	      //-----------------------------------------------------------------------------
	      // continue motion in SINGLESTEP mode
	      //-----------------------------------------------------------------------------
	      // check for execution to be waiting for new rising edge
	    ELSIF #statStateExecution = #EX_TRIGGERING_CMD
	      AND #statExecutionWaitSingleStep = TRUE
	    THEN
	      #statBusy := TRUE; // set FB state to busy
	      #statExecutionWaitSingleStep := FALSE; // reset execution wait bit stopping cmds from being executed (wait in EX_TRIGGERING_CMD)
	      //===========================================================================================
	      
	      //-----------------------------------------------------------------------------
	      // CONTINUE after interrupt
	      //-----------------------------------------------------------------------------
	      // check for path motion to be interrupted
	    ELSIF #statStateExecution = #EX_INTERRUPTED
	      OR #statStateExecution = #EX_INTERRUPTING // FR 12.10.2021
	    THEN
	      // State machine - continue path motion and sequence
	      // no changes to PreBuffer state machine
	      #statStateExecution := #EX_CONTINUEING;
	      // no setting of FB state to busy necessary, interrupt does not reset busy
	      // ==========================================================================================
	      
	      //-----------------------------------------------------------------------------
	      // RETRIGGER during running path motion
	      //-----------------------------------------------------------------------------
	      // check for path motion to be running with all previous cmds executed
	    ELSIF #statStateExecution = #EX_ALL_TRIGGERED THEN
	      #statBusy := TRUE; // set FB state to busy
	      #statLastCmdIdPathdata := 0; // reset last cmdId in PathData depending on type of attached PathData
	      #statMCExecuteWasDone := FALSE; // Reset bit to memorize done output of MC_ExecuteKinMotionCmd
	      // state machines - reStart processing
	      #statStatePreBuffering := #PB_ENABLED;
	      #statStateExecution := #EX_GET_CMD;
	      // initialize variables
	      #statReadyForNextPath := FALSE;
	      // set status - added JR 2019/04/16
	      #statStatus := #STATUS_SUBSEQUENT_CALL;
	      
	      #instLKinCtrl_PreBuffer.flagLimits.firstFlag := LOWER_BOUND(ARR := #flags, DIM := 1);
	      #instLKinCtrl_PreBuffer.flagLimits.lastFlag := UPPER_BOUND(ARR := #flags, DIM := 1);
	      
	      #instLKinCtrl_PreBuffer.flagLimits.firstValueFlag := LOWER_BOUND(ARR := #valueFlags, DIM := 1);
	      #instLKinCtrl_PreBuffer.flagLimits.lastValueFlag := UPPER_BOUND(ARR := #valueFlags, DIM := 1);
	      
	      #instLKinCtrl_MC_ExecuteKinMotionCmd.flagLimits.firstFlag := LOWER_BOUND(ARR := #flags, DIM := 1);
	      #instLKinCtrl_MC_ExecuteKinMotionCmd.flagLimits.lastFlag := UPPER_BOUND(ARR := #flags, DIM := 1);
	      
	      #instLKinCtrl_MC_ExecuteKinMotionCmd.flagLimits.firstValueFlag := LOWER_BOUND(ARR := #valueFlags, DIM := 1);
	      #instLKinCtrl_MC_ExecuteKinMotionCmd.flagLimits.lastValueFlag := UPPER_BOUND(ARR := #valueFlags, DIM := 1);
	      
	      //===========================================================================================
	      
	      //-----------------------------------------------------------------------------
	      // START of path motion (initial)
	      //-----------------------------------------------------------------------------
	      // check for path motion not to be running already
	    ELSIF #tempMotionQueueCommands = 0                      // no commands in MotionQueue
	      AND #tempKinematicsStatusWord.%X12 = TRUE             // TO Kinematics in constant velocity
	      AND #axesGroup.StatusPath.Velocity = 0.0              // TO Kinematics standing still
	      AND (#tempKinematicsStatusWord.%X6                    // no motion job in progress
	      OR #axesGroup.StatusConveyor[1].TrackingState <> 0    // If kinematics is in tracking then done (.X6) is not set
	      OR #axesGroup.StatusConveyor[2].TrackingState <> 0
	      OR #axesGroup.StatusConveyor[3].TrackingState <> 0)
	      AND #statStatus <> #STATUS_EXECUTION_WAITING          // Added FR 2019.03.28
	    THEN
	      // Initialize variables, diagnostics, etc.
	      #statStatus := #STATUS_FIRST_CALL;
	      #statStateExecution := #EX_RESETTING;
	      
	      #instLKinCtrl_PreBuffer.flagLimits.firstFlag := LOWER_BOUND(ARR := #flags, DIM := 1);
	      #instLKinCtrl_PreBuffer.flagLimits.lastFlag := UPPER_BOUND(ARR := #flags, DIM := 1);
	      
	      #instLKinCtrl_PreBuffer.flagLimits.firstValueFlag := LOWER_BOUND(ARR := #valueFlags, DIM := 1);
	      #instLKinCtrl_PreBuffer.flagLimits.lastValueFlag := UPPER_BOUND(ARR := #valueFlags, DIM := 1);
	      
	      #instLKinCtrl_MC_ExecuteKinMotionCmd.flagLimits.firstFlag := LOWER_BOUND(ARR := #flags, DIM := 1);
	      #instLKinCtrl_MC_ExecuteKinMotionCmd.flagLimits.lastFlag := UPPER_BOUND(ARR := #flags, DIM := 1);
	      
	      #instLKinCtrl_MC_ExecuteKinMotionCmd.flagLimits.firstValueFlag := LOWER_BOUND(ARR := #valueFlags, DIM := 1);
	      #instLKinCtrl_MC_ExecuteKinMotionCmd.flagLimits.lastValueFlag := UPPER_BOUND(ARR := #valueFlags, DIM := 1);
	      //===========================================================================================
	      
	    ELSE
	      //===========================================================================================
	      // Trigger not possible
	      // set execution state machine
	      #statStateExecution := #EX_ERROR_STATE;
	      #statStatus := #ERR_TRIGGER_NOT_POSSIBLE;
	      //===========================================================================================
	    END_IF;
	    
	  ELSIF (#statStatus = #STATUS_FIRST_CALL) THEN
	    #statStatus := #STATUS_SUBSEQUENT_CALL;
	  END_IF;
	  
	  // Edge detection input variables
	  #statExecuteOld := #tempExecute;
	  #statStopOld := #tempStop;
	  #statInterruptOld := #tempInterrupt;
	  #statResetOld := #tempReset;
	  
	END_REGION TRIGGERING
	
	IF (#statStatus = #STATUS_NO_CALL) THEN // Nothing to do -> End here to reduce "system load"
	  RETURN;
	END_IF;
	
	REGION RESETTING
	  IF #statStateExecution = #EX_RESETTING
	    // AND #statDebugState = TRUE
	  THEN
	    // reset  variable for single step debugging of states
	    #statDebugState := FALSE;
	    
	    // ----------------------------------------------
	    // Reset static for outputs
	    // ----------------------------------------------
	    #statDone := FALSE;
	    #statCommandAborted := FALSE;
	    #statError := FALSE;
	    #statErrorID := 16#0;
	    #statSubfunctionStatus := 16#0;
	    #diagnostics := #statEmptyDiagnostics;
	    
	    // ----------------------------------------------
	    // reset static variables
	    //-----------------------------------------------
	    #statFirstCycle := TRUE;
	    #statInterruptedAtStart := FALSE;
	    #statExecutionWaitSingleStep := FALSE;
	    #statPauseExecution := FALSE;
	    #statMCExecuteWasDone := FALSE;
	    #statPathDataIdentifier := 0;
	    #statLastCmdIdPathdata := 0;
	    #statWrittenActiveCmdNo := -1;
	    #statStoreInterruptStateExecution := 0;
	    #statPreBufferCmdCtr := "LKINCTRL_NO_OF_START_EXECUTE_CMDS";
	    #statAbortOld := FALSE;
	    #statIsMeasurementCmd := 0;
	    
	    
	    // ----------------------------------------------
	    // initialize buffer variables
	    //-----------------------------------------------
	    // Reset PathDataPreBuffered
	    #statPathDataElementPreBuffered := #statEmptyPathDataElementPreBuffered;
	    FOR #tempCtr := 1 TO "LKINCTRL_NO_OF_PATHDATA_PREBUFFER_ELEMENTS" DO
	      #statPathDataPreBuffered.commands[#tempCtr] := #statEmptyPathDataElementPreBuffered;
	    END_FOR;
	    #statPathDataPreBuffered.retrievePointer := 1;
	    #statPathDataPreBuffered.addPointer := 1;
	    #statPathDataPreBuffered.addPointerRestarted := FALSE;
	    #statPathDataPreBuffered.pathDataName := '';
	    #statPathDataPreBufferAddPointerOld := 0;
	    
	    // ----------------------------------------------
	    // initialize flag handling variables
	    //-----------------------------------------------
	    // Reset waitFlags struct
	    #statWaitFlags.waitCtr := 0;
	    FOR #tempCtr := 1 TO "LKINCTRL_NO_OF_CMD_SETFLAGS" DO
	      #statWaitFlags.waitFlag[#tempCtr] := -1;
	    END_FOR;
	    
	    // Reset waitValueFlag struct
	    #statWaitValueFlags.waitCtr := 0;
	    FOR #tempCtr := 1 TO "LKINCTRL_NO_OF_CMD_VALUEFLAGS" DO
	      #statWaitValueFlags.waitFlag[#tempCtr] := -1;
	    END_FOR;
	    
	    // Reset setFlagsBuffer variables
	    #statFlagsBuffer.writeBufferElement := 1;
	    #statSetFlagsBufferWriteBufferElement_old := 1;
	    
	    // Reset setFlagBuffer
	    FOR #tempCtr := 1 TO "LKINCTRL_NO_OF_SETFLAGS_BUFFER_ELEMENTS" DO
	      #statFlagsBuffer.bufferElement[#tempCtr] := #statEmptyFlagBufferElement;
	    END_FOR;
	    
	    // ----------------------------------------------
	    // Call instances with false
	    // ----------------------------------------------
	    #instLKinCtrl_MC_ExecuteKinMotionCmd(execute                 := FALSE,
	                                         interrupt               := FALSE,
	                                         continueMotion          := FALSE,
	                                         stopMode                := #configuration.stopMode,
	                                         interruptMode           := #configuration.interruptMode,
	                                         reset                   := FALSE,
	                                         stop                    := FALSE,
	                                         writtenActiveCmdNo      := #statWrittenActiveCmdNo,
	                                         conveyorConfiguration   := #configuration.conveyorParameter,
	                                         userFrames              := #configuration.userFrames,
	                                         workspaceZones          := #configuration.workspaceZones,
	                                         kinematicsZones         := #configuration.kinematicsZones,
	                                         pauseCmdExecution       => #statPauseExecution,
	                                         activePathDataName      => #statActivePathData,
	                                         activeCmdNo             => #statActiveCmdNo,
	                                         remainingDistanceActCmd => #statRemainingDistanceActCmd,
	                                         activeUserFrames        => #activeUserFrames,
	                                         pathDataElementPreBuf   := #statPathDataElementPreBuffered,
	                                         to_Kinematics           := #axesGroup);
	    
	    IF #statStatus = #STATUS_FB_RESETTING
	      OR #statStatus = #STATUS_FIRST_CALL
	    THEN
	      #instLKinCtrl_MC_ExecuteKinMotionCmd.reset := TRUE; // If resetting then also reset MC_ExecuteKinMotionCmd
	      #instLKinCtrl_MC_ExecuteKinMotionCmd(execute                 := FALSE,
	                                           interrupt               := FALSE,
	                                           continueMotion          := FALSE,
	                                           stopMode                := #configuration.stopMode,
	                                           interruptMode           := #configuration.interruptMode,
	                                           //reset := FALSE, // written above
	                                           stop                    := FALSE,
	                                           writtenActiveCmdNo      := #statWrittenActiveCmdNo,
	                                           conveyorConfiguration   := #configuration.conveyorParameter,
	                                           userFrames              := #configuration.userFrames,
	                                           workspaceZones          := #configuration.workspaceZones,
	                                           kinematicsZones         := #configuration.kinematicsZones,
	                                           pauseCmdExecution       => #statPauseExecution,
	                                           activePathDataName      => #statActivePathData,
	                                           activeCmdNo             => #statActiveCmdNo,
	                                           remainingDistanceActCmd => #statRemainingDistanceActCmd,
	                                           activeUserFrames        => #activeUserFrames,
	                                           pathDataElementPreBuf   := #statPathDataElementPreBuffered,
	                                           to_Kinematics           := #axesGroup);
	      #instLKinCtrl_MC_ExecuteKinMotionCmd.reset := FALSE; // Reset input
	    END_IF;
	    
	    #instLKinCtrl_PreBuffer(enable         := FALSE,
	                            error          => #statPreBufferError,
	                            pointTable     := #pointTable,
	                            to_Kinematics  := #axesGroup,
	                            pathData       := #pathData,
	                            pathDataPreBuf := #statPathDataPreBuffered);
	    
	    #instLKinCtrl_SetFlagCtrl(enable    := FALSE,
	                              waitMain  => #statWaitMain,
	                              flags     := #flags,
	                              waitFlags := #statWaitFlags);
	    
	    #instLKinCtrl_ValueFlagCtrl(enable     := FALSE,
	                                waitMain   => #statWaitValueMain,
	                                valueFlags := #valueFlags,
	                                waitFlags  := #statWaitValueFlags);
	    
	    // ----------------------------------------------
	    // Check if coming from reset or execute and handle differences
	    // ----------------------------------------------
	    IF #statStatus = #STATUS_FB_RESETTING THEN
	      // ---------------------------
	      // Coming from reset
	      // ---------------------------
	      #statReadyForNextPath := TRUE;
	      #statStateExecution := #EX_NO_PROCESSING;
	      #statStatePreBuffering := #PB_NO_PROCESSING;
	      #statStatus := #STATUS_NO_CALL;
	    ELSE
	      // ---------------------------
	      // Coming from execute
	      // ---------------------------
	      #statBusy := TRUE;
	      #statReadyForNextPath := FALSE;
	      #statStatePreBuffering := #PB_ENABLED;
	      IF #INTERRUPT_AT_START THEN
	        #statStateExecution := #EX_INTERRUPT_AT_START;
	      ELSIF #CONTINUE_AT_START THEN
	        #statStateExecution := #EX_CONTINUE_AT_START;
	      ELSE
	        #statStateExecution := #EX_GET_CMD;
	      END_IF;
	    END_IF;
	  END_IF;
	END_REGION RESETTING
	
	REGION ABORT_MEASUREMENT_CMD
	  //------------------------------------------------------------------------------------------
	  // Abort measurement command functionality 
	  //------------------------------------------------------------------------------------------
	  //check cyclically if abort input has been reset
	  IF (#statAbortOld = TRUE) AND (#tempAbortMeasurementCmd = FALSE) THEN
	    #statAbortOld := FALSE;
	    
	    //first call of abort functionality
	  ELSIF (#tempAbortMeasurementCmd = TRUE) AND (#statAbortOld = FALSE) THEN
	    IF ((#statIsMeasurementCmd = "LKINCTRL_MEAS_CMD_WO_ACK")
	      OR (#statIsMeasurementCmd = "LKINCTRL_MEAS_CMD_WITH_ACK"))
	    THEN
	      #statActiveCmdNoOld := #statActiveCmdNo;
	      #statStateOld := #statStateExecution;
	      #statStateExecution := #EX_ABORT_MEAS_CMD;
	      #statAbortOld := TRUE;
	    END_IF;
	    
	    //for multiple measurement commands in a row (1,1,1 or 1,1,1,2)
	  ELSIF (#tempAbortMeasurementCmd = TRUE) AND (#statAbortOld = TRUE) THEN
	    IF ((#statIsMeasurementCmd = "LKINCTRL_MEAS_CMD_WO_ACK") OR (#statIsMeasurementCmd = "LKINCTRL_MEAS_CMD_WITH_ACK"))
	      AND (#statActiveCmdNo = (#statActiveCmdNoOld + 1))
	    THEN
	      #statActiveCmdNoOld := #statActiveCmdNo;
	      #statStateOld := #statStateExecution;
	      #statStateExecution := #EX_ABORT_MEAS_CMD;
	      #statAbortOld := TRUE;
	    END_IF;
	  END_IF;
	END_REGION
	
	REGION PRE_BUFFERING
	  
	  // state reached when no pre buffering is active
	  REGION PB_NO_PROCESSING
	    IF #statStatePreBuffering = #PB_NO_PROCESSING
	      // AND #statDebugState = TRUE
	    THEN
	      // reset  variable for single step debugging of states
	      #statDebugState := FALSE;
	      
	      // Do nothing here
	    END_IF;
	  END_REGION PB_NO_PROCESSING
	  
	  // state reached when pre buffering is active
	  REGION PB_ENABLED
	    IF #statStatePreBuffering = #PB_ENABLED
	      // AND #statDebugState = TRUE
	    THEN
	      // reset  variable for single step debugging of states
	      #statDebugState := FALSE;
	      
	      IF #statStatus = #STATUS_FIRST_CALL THEN
	        #statInitStartPos := TRUE;
	      END_IF;
	      
	      
	      // Call FB PreBuffer multiple times
	      FOR #tempCtr := 1 TO #statPreBufferCmdCtr DO
	        
	        // Call FB PreBuffer
	        #instLKinCtrl_PreBuffer(enable                  := TRUE,
	                                initPathTransition      := #pathTransition,
	                                initBufferMode          := #bufferMode,
	                                initTransitionParameter := #transitionParameter,
	                                initStartPosition       := #statInitStartPos,
	                                configuration           := #configuration,
	                                error                   => #statPreBufferError,
	                                pointTable              := #pointTable,
	                                to_Kinematics           := #axesGroup,
	                                lastCmdIdPathData       => #statLastCmdIdPathdata,
	                                pathData                := #pathData,
	                                pathDataPreBuf          := #statPathDataPreBuffered);
	        
	        #statInitStartPos := FALSE;
	        
	        // check for FB PreBuffer to signalize an error
	        IF #statPreBufferError THEN
	          IF #instLKinCtrl_MC_ExecuteKinMotionCmd.busy THEN
	            #statStatus := #STATUS_STOP_DUE_TO_ERROR; // Error at command --> Stop Kinematics
	          ELSE
	            #statStatus := #ERR_PATHDATA_PARAMETERS;
	          END_IF;
	          #statSubfunctionStatus := #instLKinCtrl_PreBuffer.status;// Store subfunction status
	          #statStatePreBuffering := #PB_DISABLED; // Disable preBuffer
	          #statStateExecution := #EX_ERROR_STATE;
	          // Write diagnostics
	          #diagnostics.pathDataName := #statPathDataPreBuffered.pathDataName;
	          #diagnostics.cmdNumber := #instLKinCtrl_PreBuffer.pathDataRetrievePointer;
	          EXIT; // exit loop to end pre buffering
	        END_IF;
	        
	        // Check for FB PreBuffer to have buffered the last element of the PathData to PathData_PreBuf
	        IF #instLKinCtrl_PreBuffer.status = 16#7100 THEN // STATUS_ALL_CMDS_BUFFERED
	          #statStatePreBuffering := #PB_DISABLED; // go to disable state when PreBuffer is done
	          EXIT; // exit loop to end pre buffering
	        END_IF;
	        
	      END_FOR;
	    END_IF;
	  END_REGION PB_ENABLED
	  
	  // state reached when pre buffering is active
	  REGION PB_DISABLED
	    IF #statStatePreBuffering = #PB_DISABLED
	      // AND #statDebugState = TRUE
	    THEN
	      // reset  variable for single step debugging of states
	      #statDebugState := FALSE;
	      
	      // call FB_PreBuffer with false
	      // second call of FB necessary, for PathData with one command only ==> handled in one cycle only
	      #instLKinCtrl_PreBuffer(enable         := FALSE,
	                              pointTable     := #pointTable,
	                              to_Kinematics  := #axesGroup,
	                              pathData       := #pathData,
	                              pathDataPreBuf := #statPathDataPreBuffered);
	      
	    END_IF;
	  END_REGION PB_DISABLED
	  
	END_REGION PRE_BUFFERING
	
	
	REGION EXECUTION
	  // Call Execution steps multiple times
	  FOR #tempExecCtr := 1 TO #statPreBufferCmdCtr DO
	    
	    
	    // state reached when no processing is active 
	    REGION EX_NO_PROCESSING
	      IF #statStateExecution = #EX_NO_PROCESSING
	        // AND #statDebugState = TRUE
	      THEN
	        // reset  variable for single step debugging of states
	        #statDebugState := FALSE;
	        
	        // do nothing and wait for execute trigger
	      END_IF;
	    END_REGION EX_NO_PROCESSING
	    
	    REGION EX_INTERRUPT_AT_START
	      IF #statStateExecution = #EX_INTERRUPT_AT_START THEN
	        #instLKinCtrl_MC_ExecuteKinMotionCmd.interrupt := TRUE; // Simulate interrupt input
	        
	        IF #instLKinCtrl_MC_ExecuteKinMotionCmd.diagnostics.status = 16#7102 THEN // Check if interrupted
	          // Interrupted --> Start executing commands
	          #instLKinCtrl_MC_ExecuteKinMotionCmd.interrupt := FALSE;
	          #statInterruptedAtStart := TRUE;
	          #statStateExecution := #EX_GET_CMD;
	        END_IF;
	      END_IF;
	    END_REGION EX_INTERRUPT_AT_START
	    
	    REGION EX_CONTINUE_AT_START
	      // Due to a system bug up to FW4.0 (blending, override) a groupContinue must always be triggered after a groupInterrupt even if the interrupt was aborted with a groupStop.
	      // To avoid checking for aborted interrupts we always trigger continue at the start of a path.
	      IF #statStateExecution = #EX_CONTINUE_AT_START THEN
	        IF #tempKinematicsStatusWord.%X17 = FALSE THEN // Only continue if not interrupted as we dont want to trigger a movement
	          #instLKinCtrl_MC_ExecuteKinMotionCmd.continueMotion := TRUE; // Trigger continue
	          
	          IF #instLKinCtrl_MC_ExecuteKinMotionCmd.diagnostics.status = 16#7100 THEN // Check if continue is done
	            #instLKinCtrl_MC_ExecuteKinMotionCmd.continueMotion := FALSE;
	            #statStateExecution := #EX_GET_CMD;
	          END_IF;
	        ELSE
	          // Go to next step if interrupted from extern
	          #statStateExecution := #EX_GET_CMD;
	        END_IF;
	      END_IF;
	    END_REGION EX_CONTINUE_AT_START
	    
	    // state reached new command should be provided from PathData_PreBuffered to LKinCtrl_ExecuteKinMotionCmd 
	    REGION EX_GET_CMD
	      IF #statStateExecution = #EX_GET_CMD
	        // AND #statDebugState = TRUE
	      THEN
	        // reset  variable for single step debugging of states
	        #statDebugState := FALSE;
	        #statSubfunctionStatus := 16#0;
	        
	        // check for lastCmdIdPathInData to be recognized after last execution of EX_TRIGGERED_CMD
	        IF #statPathDataElementPreBuffered.cmdID = #statLastCmdIdPathdata
	          AND #statPathDataElementPreBuffered.isIntermediateCmd = FALSE
	        THEN
	          // skip GET_NEW_CMD and go to EX_ALL_TRIGGERED
	          #statStateExecution := #EX_ALL_TRIGGERED;
	        ELSE
	          // ------------------------------------------------------------------------------------------
	          // Get new cmd from PathData_PreBuffered according to the pointer status
	          // ------------------------------------------------------------------------------------------
	          // Initialize temp
	          #tempPreBufferPtrOk := FALSE;
	          
	          // Check if addPointer was restarted 
	          IF #statPathDataPreBuffered.addPointerRestarted THEN
	            // addPointer must not pass retrievePointer (no overwriting not read slots), addPointer may not pass
	            #tempPreBufferPtrOk := #statPathDataPreBuffered.retrievePointer > #statPathDataPreBuffered.addPointer;
	            
	            // Special cases in first cycle or contourOffset and addPointerRestarted
	            IF #statStatus = #STATUS_FIRST_CALL OR #instLKinCtrl_PreBuffer.preBufferLockDueToConfigCmd THEN
	              #tempPreBufferPtrOk := TRUE;
	            END_IF;
	          ELSE
	            // retrievePointer must not pass addPointer (no reading of empty slots), retrievePointer may not pass
	            #tempPreBufferPtrOk := #statPathDataPreBuffered.retrievePointer < #statPathDataPreBuffered.addPointer;
	          END_IF;
	          
	          IF #tempPreBufferPtrOk THEN
	            // ------------------------------------------------------------------------------------------
	            // Copy command for execution and increase retrievePointer
	            // ------------------------------------------------------------------------------------------
	            #statPathDataElementPreBuffered := #statPathDataPreBuffered.commands[#statPathDataPreBuffered.retrievePointer];
	            
	            // Calculate new retrievePointer
	            IF #statPathDataPreBuffered.retrievePointer < "LKINCTRL_NO_OF_PATHDATA_PREBUFFER_ELEMENTS" THEN
	              #statPathDataPreBuffered.retrievePointer += 1;
	            ELSE
	              #statPathDataPreBuffered.retrievePointer := 1;  // restart PathDataPreBuf retrievePointer
	              #statPathDataPreBuffered.addPointerRestarted := FALSE; // reset restart bit of pointer
	            END_IF;
	            
	            // ------------------------------------------------------------------------------------------
	            // PathData identifier number - setting
	            // ------------------------------------------------------------------------------------------
	            // detect change of PathData - new cmdId smaller or equal to last one ==> new Path
	            IF (#statPathDataElementPreBuffered.cmdID <= #statPreBufferedCmdIdOld)
	              OR (#statPathDataElementPreBuffered.pathDataName <> #statPreBufferedPathDataNameOld)
	            THEN
	              // handle PathData identifier counter
	              IF #statPathDataIdentifier < "LKINCTRL_NO_OF_SETFLAGS_BUFFER_ELEMENTS" THEN
	                #statPathDataIdentifier += 1; // increase PathData counter
	              ELSE
	                #statPathDataIdentifier := 1; // restart PathData identifier counter
	              END_IF;
	            END_IF;
	            
	            // write PathData identifier in PatDataElement_preBuffered
	            #statPathDataElementPreBuffered.pathDataIdentifier := #statPathDataIdentifier;
	            
	            // store old cmdID and PathDataName
	            #statPreBufferedCmdIdOld := #statPathDataElementPreBuffered.cmdID;
	            #statPreBufferedPathDataNameOld := #statPathDataElementPreBuffered.pathDataName;
	            
	            
	            // ------------------------------------------------------------------------------------------
	            // FLAG information - store and evaluate
	            // ------------------------------------------------------------------------------------------
	            // copy command setFlags for storing and usage in flag handling
	            // setFlagsBuffer has twice the number of slots of PathDataPreBuffered to store flag information of past executed (already in MotionQueue) commands
	            #tempFlagBufferElement.pathDataName := #statPathDataElementPreBuffered.pathDataName;
	            #tempFlagBufferElement.pathDataIdentifier := #statPathDataIdentifier;
	            #tempFlagBufferElement.cmdId := #statPathDataElementPreBuffered.cmdID;
	            #tempFlagBufferElement.setFlags := #statPathDataElementPreBuffered.setFlags;
	            #tempFlagBufferElement.valueFlags := #statPathDataElementPreBuffered.valueFlags;
	            #tempFlagBufferElement.isIntermediateCmd := #statPathDataElementPreBuffered.isIntermediateCmd;
	            
	            #statFlagsBuffer.bufferElement[#statFlagsBuffer.writeBufferElement] := #tempFlagBufferElement;
	            
	            #statSetFlagsBufferWriteBufferElement_old := #statFlagsBuffer.writeBufferElement;
	            
	            // increase statSetFlagsBuffer write pointer and restart at overflow
	            IF #statFlagsBuffer.writeBufferElement < "LKINCTRL_NO_OF_SETFLAGS_BUFFER_ELEMENTS" THEN
	              #statFlagsBuffer.writeBufferElement := #statFlagsBuffer.writeBufferElement + 1;
	            ELSE
	              #statFlagsBuffer.writeBufferElement := 1;
	            END_IF;
	            
	            // ------------------------------------------------------------------------------------------
	            // Go to next state --> Trigger command
	            // ------------------------------------------------------------------------------------------
	            #statStateExecution := #EX_TRIGGERING_CMD;
	            
	          ELSE
	            // ------------------------------------------------------------------------------------------
	            // PreBuffer Pointer do not allow for next command
	            // ------------------------------------------------------------------------------------------ 
	            // set subfunction status according to PreBuffer status
	            IF (#statPathDataPreBuffered.retrievePointer = #statPathDataPreBuffered.addPointer
	              AND #statPathDataPreBuffered.addPointerRestarted = FALSE)
	            THEN
	              #statSubfunctionStatus := #STATUS_WAITING_FOR_PREBUFFERED_CMD;
	              
	            ELSIF (#statPathDataPreBuffered.addPointerRestarted = TRUE
	              AND (#statPathDataPreBuffered.retrievePointer - 1 = #statPathDataPreBuffered.addPointer))
	            THEN
	              #statSubfunctionStatus := #STATUS_PREBUFFERED_FULL;
	            END_IF;
	            
	          END_IF;
	          
	          // ------------------------------------------------------------------------------------------
	          // Check if interrupt was executed at start and if continue is needed
	          // ------------------------------------------------------------------------------------------
	          IF #statInterruptedAtStart THEN
	            IF #tempMotionQueueCommands >= MIN(IN1 := #NO_OF_COMMANDS_PRELOADING, IN2 := #axesGroup.MotionQueue.MaxNumberOfCommands)
	              OR #statPauseExecution // Continue if FB ExecuteKinMotionCmd signalizes pause else we have a deadlock
	              OR #statPathDataElementPreBuffered.cmdID = #statLastCmdIdPathdata // Continue if end of path was reached
	            THEN
	              #statStoreInterruptStateExecution := #statStateExecution;
	              #statStateExecution := #EX_CONTINUEING;
	              #statInterruptedAtStart := FALSE;
	            END_IF;
	          END_IF;
	        END_IF;
	      END_IF;
	    END_REGION EX_GET_CMD
	    
	    
	    // state reached when cmd should be triggered
	    REGION EX_TRIGGERING_CMD
	      IF #statStateExecution = #EX_TRIGGERING_CMD
	        // AND #statDebugState = TRUE
	      THEN
	        // Reset variable for single step debugging of states
	        #statDebugState := FALSE;
	        
	        // Create condition for execution
	        #tempExecutionWaiting := #statExecutionWaitSingleStep OR #statPauseExecution OR #statWaitMain OR #statWaitValueMain;
	        
	        IF #tempExecutionWaiting = FALSE THEN
	          // ------------------------------------------------------------------------------------------
	          // Trigger FB_ExecutePathMotion to execute cmd in same cycle
	          // ------------------------------------------------------------------------------------------ 
	          #instLKinCtrl_MC_ExecuteKinMotionCmd.execute := TRUE;
	        ELSIF #instLKinCtrl_MC_ExecuteKinMotionCmd.active = FALSE AND #statStatus <> #STATUS_CMD_CONFIGURATION_ACTIVE AND #tempMotionQueueCommands = 0 THEN
	          // ------------------------------------------------------------------------------------------ 
	          // Execution is waiting
	          // ------------------------------------------------------------------------------------------  
	          #statStatus := #STATUS_EXECUTION_WAITING;
	        ELSE
	          ;
	        END_IF;
	      END_IF;
	    END_REGION EX_TRIGGERING_CMD
	    
	    // state reached when GroupInterrupt is interrupted ==> do nothing when interrupted
	    REGION EX_CONTINUEING
	      IF #statStateExecution = #EX_CONTINUEING
	        // AND #statDebugState = TRUE
	      THEN
	        // reset  variable for single step debugging of states
	        #statDebugState := FALSE;
	        
	        // FR 14.12.2021: Switched IF and trigger to at least have one cycle where continueMotion is true
	        
	        // set state machine to CONTINUED after successfull continue of path motion
	        IF #instLKinCtrl_MC_ExecuteKinMotionCmd.diagnostics.status = 16#7100 // Motion was continued
	          OR (#statMCExecuteWasDone = TRUE AND #instLKinCtrl_MC_ExecuteKinMotionCmd.continueMotion = TRUE) // Motion was done but continue was triggered at least for one cycle
	        THEN
	          #statStateExecution := #EX_CONTINUED;
	        END_IF;
	        
	        // set continueMotion input on LKinCtrl_ExecuteKinMotionCmd
	        // FR 12.10.2021
	        #instLKinCtrl_MC_ExecuteKinMotionCmd.execute := FALSE; // Reset execute
	        #instLKinCtrl_MC_ExecuteKinMotionCmd.continueMotion := TRUE; // Trigger continue
	        #instLKinCtrl_MC_ExecuteKinMotionCmd.interrupt := FALSE; // Reset interrupt
	        
	      END_IF;
	    END_REGION EX_CONTINUEING
	    
	    
	    // state reached when GroupContinue is done ==> do nothing when path motion continues
	    REGION EX_CONTINUED
	      IF #statStateExecution = #EX_CONTINUED
	        // AND #statDebugState = TRUE
	      THEN
	        // reset  variable for single step debugging of states
	        #statDebugState := FALSE;
	        
	        #instLKinCtrl_MC_ExecuteKinMotionCmd.continueMotion := FALSE; // reset continueMotion input on LKinCtrl_ExecuteKinMotionCmd
	        #statStatus := #STATUS_PATHMOTION_RUNNING; // set status accordingly
	        #statStateExecution := #statStoreInterruptStateExecution; // set state machine to state before interrupt
	      END_IF;
	    END_REGION EX_CONTINUED
	    
	    // state reached to execute MC_GroupInterrupt ==> wait for interrupt to be done
	    REGION EX_INTERRUPTING
	      IF #statStateExecution = #EX_INTERRUPTING
	        // AND #statDebugState = TRUE
	      THEN
	        // reset  variable for single step debugging of states
	        #statDebugState := FALSE;
	        
	        #instLKinCtrl_MC_ExecuteKinMotionCmd.execute := FALSE; // Reset execute
	        #instLKinCtrl_MC_ExecuteKinMotionCmd.continueMotion := FALSE; // FR 11.03.2020: Also reset continue input
	        #instLKinCtrl_MC_ExecuteKinMotionCmd.interrupt := TRUE; // Trigger interrupt
	        
	        // check for path motion to have been interrupted (by LKinCtrlExecuteKinMotionCmd)
	        IF #instLKinCtrl_MC_ExecuteKinMotionCmd.diagnostics.status = 16#7102 THEN
	          #statStateExecution := #EX_INTERRUPTED;
	        END_IF;
	      END_IF;
	    END_REGION EX_INTERRUPTING
	    
	    
	    // state reached when path motion has been interrupted in LKinExectuteKinMotionCmd
	    REGION EX_INTERRUPTED
	      IF #statStateExecution = #EX_INTERRUPTED
	        // AND #statDebugState = TRUE
	      THEN
	        // reset variable for single step debugging of states
	        #statDebugState := FALSE;
	        
	        #instLKinCtrl_MC_ExecuteKinMotionCmd.interrupt := FALSE; // Reset interrupt input
	        #statStatus := #STATUS_PATHMOTION_INTERRUPTED; // set status accordingly
	      END_IF;
	    END_REGION EX_INTERRUPTED
	    
	    REGION EX_ABORT_MEAS_CMD
	      IF #statStateExecution = #EX_ABORT_MEAS_CMD
	        //AND #statDebugState = TRUE
	      THEN
	        //abort command
	        #tempStopMeasure := TRUE;
	        #instLKinCtrl_MC_ExecuteKinMotionCmd.execute := FALSE; // Reset execute
	        #instLKinCtrl_MC_ExecuteKinMotionCmd.continueMotion := FALSE; // Reset continue input
	        #instLKinCtrl_MC_ExecuteKinMotionCmd.interrupt := FALSE; // Reset interrupt
	        
	        #statStatus := #STATUS_PATHMOTION_STOPPING; // set status accordingly
	        
	        IF #instLKinCtrl_MC_ExecuteKinMotionCmd.commandAborted THEN // check for path motion to be aborted in LKinExectuteKinMotionCmd
	          #statStateExecution := #EX_MEAS_CMD_ABORTED;
	          #tempStopMeasure := FALSE;
	        ELSIF #instLKinCtrl_MC_ExecuteKinMotionCmd.diagnostics.status.%X15 THEN // check for executer status >= 16#8000
	          #statStateExecution := #EX_ERROR_STATE;
	          #statStatus := #ERR_EXECUTE_KINMOTIONCMD;
	          #statSubfunctionStatus := #instLKinCtrl_MC_ExecuteKinMotionCmd.diagnostics.status;
	        END_IF;
	        
	      END_IF;
	    END_REGION EX_ABORT_MEAS_CMD
	    
	    REGION EX_MEAS_CMD_ABORTED
	      IF #statStateExecution = #EX_MEAS_CMD_ABORTED THEN
	        //if abort signal has to be acknowledged in order to continue
	        IF #statIsMeasurementCmd = "LKINCTRL_MEAS_CMD_WITH_ACK" THEN
	          IF #tempAbortMeasurementCmd = FALSE THEN
	            #statAbortOld := FALSE;
	            #statStateExecution := #statStateOld;
	            IF #statStateExecution = #EX_ALL_TRIGGERED THEN
	              #statMCExecuteWasDone := TRUE;
	            END_IF;
	          END_IF;
	        ELSIF #statIsMeasurementCmd = "LKINCTRL_MEAS_CMD_WO_ACK" THEN
	          #statStateExecution := #statStateOld;
	          IF #statStateExecution = #EX_ALL_TRIGGERED THEN
	            #statMCExecuteWasDone := TRUE;
	          END_IF;
	          IF #tempAbortMeasurementCmd = FALSE THEN
	            #statAbortOld := FALSE;
	          END_IF;
	        END_IF;
	      END_IF;
	    END_REGION EX_MEAS_CMD_ABORTED
	    
	    // state reached when stop input is triggered (path motion stop is executed in LKinExectuteKinMotionCmd)
	    REGION EX_STOPPING
	      IF #statStateExecution = #EX_STOPPING
	        // AND #statDebugState = TRUE
	      THEN
	        // reset variable for single step debugging of states
	        #statDebugState := FALSE;
	        
	        #instLKinCtrl_MC_ExecuteKinMotionCmd.execute := FALSE; // Reset execute
	        #instLKinCtrl_MC_ExecuteKinMotionCmd.continueMotion := FALSE; // Reset continue input
	        #instLKinCtrl_MC_ExecuteKinMotionCmd.interrupt := FALSE; // Reset interrupt
	        
	        #statStatus := #STATUS_PATHMOTION_STOPPING; // set status accordingly
	        
	        IF #instLKinCtrl_MC_ExecuteKinMotionCmd.commandAborted THEN // check for path motion to be aborted in LKinExectuteKinMotionCmd
	          #statStateExecution := #EX_STOPPED_STATE;
	        ELSIF #instLKinCtrl_MC_ExecuteKinMotionCmd.diagnostics.status.%X15 THEN // check for executer status >= 16#8000
	          #statStateExecution := #EX_ERROR_STATE;
	          #statStatus := #ERR_EXECUTE_KINMOTIONCMD;
	          #statSubfunctionStatus := #instLKinCtrl_MC_ExecuteKinMotionCmd.diagnostics.status;
	        END_IF;
	      END_IF;
	    END_REGION EX_STOPPING
	    
	    // state reached when path motion has been stopped in LKinExectuteKinMotionCmd
	    REGION EX_STOPPED_STATE
	      IF #statStateExecution = #EX_STOPPED_STATE
	        // AND #statDebugState = TRUE
	      THEN
	        // reset  variable for single step debugging of states
	        #statDebugState := FALSE;
	        
	        // set status accordingly
	        #statStatus := #STATUS_COMMAND_ABORTED;
	        #statSubfunctionStatus := #instLKinCtrl_MC_ExecuteKinMotionCmd.diagnostics.status;
	        
	        //------------------------------------------------------------------------------------------
	        // added 2020.02.07 DF: call Prebuffer with false (reset retrievePointer)
	        #instLKinCtrl_PreBuffer(enable         := FALSE,
	                                pointTable     := #pointTable,
	                                to_Kinematics  := #axesGroup,
	                                pathData       := #pathData,
	                                pathDataPreBuf := #statPathDataPreBuffered);
	        //------------------------------------------------------------------------------------------
	        // do nothing, wait in this state
	        
	      END_IF;
	    END_REGION EX_STOPPED_STATE
	    
	    
	    // state reached when error occured
	    REGION EX_ERROR_STATE
	      IF #statStateExecution = #EX_ERROR_STATE
	        // AND #statDebugState = TRUE
	      THEN
	        // reset  variable for single step debugging of states
	        #statDebugState := FALSE;
	        
	        // ------------------------------------------------------
	        // Reset inputs of FB MC_ExecuteKinMotionCmd
	        // ------------------------------------------------------
	        #instLKinCtrl_MC_ExecuteKinMotionCmd.execute := FALSE; // Reset execute
	        #instLKinCtrl_MC_ExecuteKinMotionCmd.continueMotion := FALSE; // Reset continue input
	        #instLKinCtrl_MC_ExecuteKinMotionCmd.interrupt := FALSE; // Reset interrupt
	        
	        // ------------------------------------------------------
	        // Check FB MC_ExecuteKinMotionCmd for error
	        // ------------------------------------------------------
	        IF #instLKinCtrl_MC_ExecuteKinMotionCmd.error THEN
	          // set status accordingly
	          IF #statSubfunctionStatus = 16#8245 // Error at Kinematics --> Nothing more to do
	            OR #statSubfunctionStatus = 16#8244  // Error GroupStop failed --> Nothing more to do
	          THEN
	            #statStatus := #ERR_EXECUTE_KINMOTIONCMD;
	          ELSE
	            #statStatus := #STATUS_STOP_DUE_TO_ERROR; // Error at command --> Stop Kinematics
	          END_IF;
	        END_IF;
	        
	        // ------------------------------------------------------
	        // Set error status if stop was successful
	        // ------------------------------------------------------
	        IF #statStatus = #STATUS_STOP_DUE_TO_ERROR AND #instLKinCtrl_MC_ExecuteKinMotionCmd.commandAborted THEN
	          IF #statPreBufferError THEN
	            // Error was caused by FB Prebuffer
	            // separate handling for PathData malconfiguration and offset compensation calculation errors
	            IF #statSubfunctionStatus > 16#8300 AND #statSubfunctionStatus <= 16#8320 THEN
	              #statStatus := #ERR_OFFSET_CALCULATION; // write status information to be error in offset compensation
	            ELSE
	              #statStatus := #ERR_PATHDATA_PARAMETERS; // write status information to be malparametrization in PathData (no offset compensation)
	            END_IF;
	          ELSE
	            // Error was caused by FB MC_ExecuteKinMotionCmd
	            #statStatus := #ERR_EXECUTE_KINMOTIONCMD;
	          END_IF;
	        END_IF;
	        
	        // ------------------------------------------------------
	        // Check if stop also failed with error
	        // ------------------------------------------------------
	        IF #instLKinCtrl_MC_ExecuteKinMotionCmd.stop AND #instLKinCtrl_MC_ExecuteKinMotionCmd.error THEN
	          #statStatus := #ERR_EXECUTE_KINMOTIONCMD;
	        END_IF;
	        
	        // ------------------------------------------------------
	        // Trigger stop input of FB MC_ExecuteKinMotionCmd
	        // ------------------------------------------------------
	        IF #statStatus = #STATUS_STOP_DUE_TO_ERROR THEN
	          #tempStop := TRUE;
	        END_IF;
	        
	      END_IF;
	    END_REGION EX_ERROR_STATE
	    
	    
	    
	    REGION CALL_FB_EXECUTE_CYCLIC
	      IF #statStatus <> #STATUS_NO_CALL THEN
	        //------------------------------------------------------------------------------------------
	        // Call FB LKinCtrl_ExecuteKinMotionCmd in every cycle to keep FB outputs updated
	        //------------------------------------------------------------------------------------------
	        // execute: set in EX_TRIGGERING_CMD
	        // interrupt: set in EX_INTERRUPTING
	        // continue: set in EX_CONTINUEING
	        #instLKinCtrl_MC_ExecuteKinMotionCmd(//execute := FALSE,
	                                             //interrupt := FALSE
	                                             //continueMotion := FALSE,
	                                             stop                    := (#tempStop OR #tempStopMeasure),
	                                             stopMode                := #configuration.stopMode,
	                                             interruptMode           := #configuration.interruptMode,
	                                             writtenActiveCmdNo      := #statWrittenActiveCmdNo,
	                                             conveyorConfiguration   := #configuration.conveyorParameter,
	                                             userFrames              := #configuration.userFrames,
	                                             workspaceZones          := #configuration.workspaceZones,
	                                             kinematicsZones         := #configuration.kinematicsZones,
	                                             pauseCmdExecution       => #statPauseExecution,
	                                             activePathDataName      => #statActivePathData,
	                                             activeCmdNo             => #statActiveCmdNo,
	                                             remainingDistanceActCmd => #statRemainingDistanceActCmd,
	                                             isMeasurementCmd        => #statIsMeasurementCmd,
	                                             activeUserFrames        => #activeUserFrames,
	                                             pathDataElementPreBuf   := #statPathDataElementPreBuffered,
	                                             to_Kinematics           := #axesGroup);
	        
	        //------------------------------------------------------------------------------------------
	        // Check outputs of FB LKinCtrl_ExecuteKinMotionCmd
	        //------------------------------------------------------------------------------------------
	        //----------------------------
	        // Done
	        //----------------------------
	        IF #instLKinCtrl_MC_ExecuteKinMotionCmd.done THEN
	          #statMCExecuteWasDone := TRUE; // Store done in separate variable for wait flag handling
	          //#instLKinCtrl_PreBuffer.preprocessingStop := FALSE; // Reset preprocessing stop for LKinLang
	        END_IF;
	        
	        //----------------------------
	        // Busy
	        //----------------------------
	        IF #instLKinCtrl_MC_ExecuteKinMotionCmd.busy THEN
	          #statMCExecuteWasDone := FALSE;
	        END_IF;
	        
	        //----------------------------
	        // Error
	        //----------------------------
	        IF #instLKinCtrl_MC_ExecuteKinMotionCmd.error THEN
	          #statSubfunctionStatus := #instLKinCtrl_MC_ExecuteKinMotionCmd.diagnostics.status;// Store error in subfunction state
	          #statStateExecution := #EX_ERROR_STATE; // set state machine to error state
	          // Write diagnostics
	          #diagnostics.motionFBStatus := #instLKinCtrl_MC_ExecuteKinMotionCmd.diagnostics.motionFBstatus;
	          #diagnostics.motionFBNumber := #instLKinCtrl_MC_ExecuteKinMotionCmd.diagnostics.faultFBNumber;
	          #diagnostics.pathDataName := #instLKinCtrl_MC_ExecuteKinMotionCmd.diagnostics.faultPathDataName;
	          #diagnostics.cmdNumber := #instLKinCtrl_MC_ExecuteKinMotionCmd.diagnostics.faultSetNumber;
	          #diagnostics.kinematicsErrorWord := #instLKinCtrl_MC_ExecuteKinMotionCmd.diagnostics.kinematicsErrorWord;
	        END_IF;
	        
	        //----------------------------
	        // External stop (#status=16#7103)
	        //----------------------------
	        IF #instLKinCtrl_MC_ExecuteKinMotionCmd.diagnostics.status = 16#7103 // Executer is stopping
	          AND #statStatus.%X15 = FALSE // MovePath has no error
	          AND #statStatus <> #STATUS_STOP_DUE_TO_ERROR // MovePath is not stopping due to error
	          AND #statStateExecution <> #EX_ABORT_MEAS_CMD
	          AND #statStateExecution <> #EX_MEAS_CMD_ABORTED
	        THEN
	          // set status accordingly
	          #statStateExecution := #EX_STOPPING;
	          #statStatus := #STATUS_PATHMOTION_STOPPING;
	          #statSubfunctionStatus := #instLKinCtrl_MC_ExecuteKinMotionCmd.diagnostics.status;
	        END_IF;
	        
	        //----------------------------
	        // CmdExecuted
	        //----------------------------
	        IF #instLKinCtrl_MC_ExecuteKinMotionCmd.cmdExecuted THEN
	          IF #statStateExecution = #EX_TRIGGERING_CMD THEN
	            #statStateExecution := #EX_TRIGGERED_CMD; // go to state triggered when command has been successfully executed to MotionQueue
	          END_IF;
	        END_IF;
	        
	        //------------------------------------------------------------------------------------------
	        // Call FB LKinCtrl_ExecuteKinMotionCmd with execute := FALSE to create new rising edge
	        //------------------------------------------------------------------------------------------
	        IF #instLKinCtrl_MC_ExecuteKinMotionCmd.cmdExecuted OR #instLKinCtrl_MC_ExecuteKinMotionCmd.done THEN
	          #instLKinCtrl_MC_ExecuteKinMotionCmd(execute                 := FALSE,
	                                               stop                    := (#tempStop OR #tempStopMeasure),
	                                               stopMode                := #configuration.stopMode,
	                                               interruptMode           := #configuration.interruptMode,
	                                               writtenActiveCmdNo      := #statWrittenActiveCmdNo,
	                                               conveyorConfiguration   := #configuration.conveyorParameter,
	                                               userFrames              := #configuration.userFrames,
	                                               workspaceZones          := #configuration.workspaceZones,
	                                               kinematicsZones         := #configuration.kinematicsZones,
	                                               pauseCmdExecution       => #statPauseExecution,
	                                               activePathDataName      => #statActivePathData,
	                                               activeCmdNo             => #statActiveCmdNo,
	                                               remainingDistanceActCmd => #statRemainingDistanceActCmd,
	                                               activeUserFrames        => #activeUserFrames,
	                                               pathDataElementPreBuf   := #statPathDataElementPreBuffered,
	                                               to_Kinematics           := #axesGroup);
	          
	          //If done is set with the second call if mc executer then we could miss this here
	          //So we check for done here also
	          IF #instLKinCtrl_MC_ExecuteKinMotionCmd.done THEN
	            #statMCExecuteWasDone := TRUE;
	          END_IF;
	          
	        END_IF;
	        
	      END_IF;
	    END_REGION CALL_FB_EXECUTE_CYCLIC
	    
	    
	    // state reached when cmd has been triggered and is executed to the MotionQueue
	    REGION EX_TRIGGERED_CMD
	      IF #statStateExecution = #EX_TRIGGERED_CMD
	        // AND #statDebugState = TRUE
	      THEN
	        // reset  variable for single step debugging of states
	        #statDebugState := FALSE;
	        
	        // ------------------------------------------------------------------------------------------ 
	        // Evaluate flag information for wait flags
	        // ------------------------------------------------------------------------------------------ 
	        #tempFlagBufferElement := #statFlagsBuffer.bufferElement[#statSetFlagsBufferWriteBufferElement_old]; // Copy array element to temp
	        
	        #tempWaitFlagFound := FALSE; // Reset bit
	        
	        IF #tempFlagBufferElement.cmdId <> 0 THEN // check for cmdId not to exceed array limits
	          // run through all setFlags in command
	          FOR #tempCtr := 1 TO "LKINCTRL_NO_OF_CMD_SETFLAGS" DO
	            // check preBuffered command for wait flag
	            IF #tempFlagBufferElement.setFlags[#tempCtr].flag > -1
	              AND (#tempFlagBufferElement.setFlags[#tempCtr].flagMode = "LKINCTRL_FM_SET_BEFORE_AND_NO_RESET_AND_WAIT_FOR_ACKNOWLEDGE"
	              OR #tempFlagBufferElement.setFlags[#tempCtr].flagMode = "LKINCTRL_FM_SET_AFTER_AND_NO_RESET_AND_WAIT_FOR_ACKNOWLEDGE"
	              OR #tempFlagBufferElement.setFlags[#tempCtr].flagMode = "LKINCTRL_FM_NO_SET_AND_WAIT_FOR_FALSE_ONCE"
	              OR #tempFlagBufferElement.setFlags[#tempCtr].flagMode = "LKINCTRL_FM_NO_SET_AND_WAIT_FOR_TRUE_ONCE")
	            THEN
	              // increase counter to count activated wait flags in command
	              #statWaitFlags.waitCtr += 1;
	              // store information on which flags are wait flags
	              #statWaitFlags.waitFlag[#tempCtr] := #tempFlagBufferElement.setFlags[#tempCtr].flag;
	              #tempWaitFlagFound := TRUE; // Set bit true to exit loop
	            END_IF;
	          END_FOR;
	          
	          // run through all valueFlags in command
	          FOR #tempCtr := 1 TO "LKINCTRL_NO_OF_CMD_VALUEFLAGS" DO
	            // check preBuffered command for wait flag
	            IF #tempFlagBufferElement.valueFlags[#tempCtr].flag > -1
	              AND (#tempFlagBufferElement.valueFlags[#tempCtr].flagMode = "LKINCTRL_FM_SET_BEFORE_AND_NO_RESET_AND_WAIT_FOR_ACKNOWLEDGE"
	              OR #tempFlagBufferElement.valueFlags[#tempCtr].flagMode = "LKINCTRL_FM_SET_AFTER_AND_NO_RESET_AND_WAIT_FOR_ACKNOWLEDGE"
	              OR #tempFlagBufferElement.valueFlags[#tempCtr].flagMode = "LKINCTRL_FM_NO_SET_AND_WAIT_FOR_FALSE_ONCE"
	              OR #tempFlagBufferElement.valueFlags[#tempCtr].flagMode = "LKINCTRL_FM_NO_SET_AND_WAIT_FOR_TRUE_ONCE")
	            THEN
	              // increase counter to count activated wait value flags in command
	              #statWaitValueFlags.waitCtr += 1;
	              // store information on which flags are wait value flags
	              #statWaitValueFlags.waitFlag[#tempCtr] := #tempFlagBufferElement.valueFlags[#tempCtr].flag;
	              #tempWaitFlagFound := TRUE; // Set bit true to exit loop
	            END_IF;
	          END_FOR;
	        END_IF;
	        
	        // ------------------------------------------------------------------------------------------ 
	        // Overwrite status after ExecutionWaiting for correct flag behavior
	        // ------------------------------------------------------------------------------------------ 
	        IF #statStatus = #STATUS_EXECUTION_WAITING THEN
	          #statStatus := #STATUS_SUBSEQUENT_CALL; // Status is only active until StatusWord of kinematics overwrites it again
	        END_IF;
	        
	        // ------------------------------------------------------------------------------------------
	        // Check for executed cmd to be last cmd in PathData
	        // ------------------------------------------------------------------------------------------
	        IF #statPathDataElementPreBuffered.cmdID = #statLastCmdIdPathdata
	          AND #statPathDataElementPreBuffered.isIntermediateCmd = FALSE
	        THEN
	          #statStateExecution := #EX_ALL_TRIGGERED; // go to state to wait for done / retriggering (no further cmds to be triggered)
	        ELSE
	          #statStateExecution := #EX_GET_CMD; // go to EX_GET_CMD to get next command
	        END_IF;
	      END_IF;
	    END_REGION EX_TRIGGERED_CMD
	    
	    
	    // state reached when all cmds have been executed to the MotionQueue (wait for done or reTriggering)
	    REGION EX_ALL_TRIGGERED
	      IF #statStateExecution = #EX_ALL_TRIGGERED
	        // AND #statDebugState = TRUE
	      THEN
	        // reset  variable for single step debugging of states
	        #statDebugState := FALSE;
	        
	        // ------------------------------------------------------------------------------------------
	        // set status and status bit to set readyForNextPath output
	        // ------------------------------------------------------------------------------------------
	        #statReadyForNextPath := TRUE;
	        IF #instLKinCtrl_MC_ExecuteKinMotionCmd.activeCmdNo = #statLastCmdIdPathdata
	          AND #statPauseExecution = TRUE
	        THEN
	          #statStatus := #STATUS_EXECUTION_WAITING; // waitTime running as last cmd
	        ELSE
	          #statStatus := #STATUS_READYFORNEXTPATH;
	        END_IF;
	        
	        // ------------------------------------------------------------------------------------------
	        // Check if execution is done or waiting
	        // ------------------------------------------------------------------------------------------
	        IF #statMCExecuteWasDone // Done of ExecuteKinMotionCmd (end of PathData reached)
	          OR #statLastCmdIdPathdata = 0 // Empty PathData
	        THEN
	          IF #statWaitMain OR #statWaitValueMain THEN // Wait until all setFlags and valueFlags are acknowledged
	            #statStatus := #STATUS_EXECUTION_WAITING; // Set status to waiting until all wait flags are acknowledged
	          ELSE
	            #statStatus := #STATUS_EXECUTION_FINISHED; // Set status to set done output according to FB template
	          END_IF;
	        END_IF;
	      END_IF;
	    END_REGION EX_ALL_TRIGGERED
	    
	    
	    // ------------------------------------------------------------------------------------------
	    // Check if for loop can be continued or needs to be exited
	    // ------------------------------------------------------------------------------------------
	    IF #statStateExecution = #EX_GET_CMD
	      AND #statSubfunctionStatus <> #STATUS_WAITING_FOR_PREBUFFERED_CMD
	      AND #statSubfunctionStatus <> #STATUS_PREBUFFERED_FULL
	      AND NOT #tempWaitFlagFound // Wait flag or value flag found
	      AND #tempSequenceMode <> 1 // SingleStep off
	    THEN
	      ; // Continue for loop -> Regular get cmd without prebuffer being full
	    ELSE
	      EXIT; // Exit loop to save time
	    END_IF;
	  END_FOR;
	  
	  // set number of calls for PreBuffer & Execution
	  #statPreBufferCmdCtr := "LKINCTRL_NO_OF_SEQ_EXECUTE_CMDS";
	END_REGION EXECUTION
	
	
	REGION MOTION_STATUS
	  // set status in case no specific status has been set before
	  IF #statStatus.%X15 = FALSE THEN // no error deteceted 
	    CASE #statStatus OF
	        // Regular status that can be overwritten
	      #STATUS_SUBSEQUENT_CALL,
	      #STATUS_PATHMOTION_RUNNING,
	      #STATUS_CMD_LIN_ACTIVE,
	      #STATUS_CMD_CIRC_ACTIVE,
	      #STATUS_CMD_MOVE_DIRECT_ACTIVE,
	      #STATUS_CMD_CONFIGURATION_ACTIVE,
	      #STATUS_EXECUTION_WAITING:
	        IF #tempKinematicsStatusWord.%X8 THEN // check for linear command to be active 
	          #statStatus := #STATUS_CMD_LIN_ACTIVE;
	        ELSIF #tempKinematicsStatusWord.%X9 THEN // check for circular command to be active
	          #statStatus := #STATUS_CMD_CIRC_ACTIVE;
	        ELSIF #tempKinematicsStatusWord.%X11 THEN // check for move direct command to be active
	          #statStatus := #STATUS_CMD_MOVE_DIRECT_ACTIVE;
	        ELSIF #instLKinCtrl_MC_ExecuteKinMotionCmd.diagnostics.status = 16#7113 THEN // Configuration command active
	          #statStatus := #STATUS_CMD_CONFIGURATION_ACTIVE;
	        ELSIF (#statPauseExecution OR #statWaitMain OR #statWaitValueMain) AND #tempMotionQueueCommands = 0 THEN // Check if waiting for FB ExecuteKinMotionCmd
	          #statStatus := #STATUS_EXECUTION_WAITING;
	        ELSIF #statStatus = #STATUS_EXECUTION_WAITING THEN // Avoid overwriting waiting status with regular subsequent call
	          ;
	        ELSE // None of the above  
	          #statStatus := #STATUS_SUBSEQUENT_CALL;
	        END_IF;
	        
	      ELSE // Every other status is defined and should not be overwritten
	        ;
	    END_CASE;
	  END_IF;
	  
	END_REGION MOTION_STATUS
	
	REGION FLAG_HANDLING
	  // Call FlagHandling FBs
	  //------------------------------------------------------------------------------------------
	  // FR 16.03.2020: Reworked Flag FBs
	  // Enable flag FBs when not finished and not no call (resetting)
	  IF #statStatus = #STATUS_FIRST_CALL OR #statStatus = #STATUS_SUBSEQUENT_CALL OR #statFirstCycle THEN
	    #instLKinCtrl_SetFlagCtrl.enable := TRUE;
	    #instLKinCtrl_ValueFlagCtrl.enable := TRUE;
	  ELSIF #statStatus = #STATUS_EXECUTION_FINISHED OR #statStatus = #STATUS_NO_CALL THEN
	    #instLKinCtrl_SetFlagCtrl.enable := FALSE;
	    #instLKinCtrl_ValueFlagCtrl.enable := FALSE;
	  ELSE
	    ;
	  END_IF;
	  
	  // Boolean Flags
	  #instLKinCtrl_SetFlagCtrl(activeCmdNo              := #statActiveCmdNo,
	                            activePathDataIdentifier := #instLKinCtrl_MC_ExecuteKinMotionCmd.activePathDataIdentifier,
	                            activePathDataName       := #instLKinCtrl_MC_ExecuteKinMotionCmd.activePathDataName,
	                            remainingDistanceActCmd  := #statRemainingDistanceActCmd,
	                            kinematicsStatusWord     := #tempKinematicsStatusWord,
	                            movePathStatus           := #statStatus,
	                            flagsBuffer              := #statFlagsBuffer,
	                            waitMain                 => #statWaitMain,
	                            flags                    := #flags,
	                            waitFlags                := #statWaitFlags);
	  
	  // Check if flag control FB has thrown an error
	  IF #instLKinCtrl_SetFlagCtrl.error THEN
	    #statStatus := #ERR_SET_FLAG_CONTROL;
	    #statSubfunctionStatus := #instLKinCtrl_SetFlagCtrl.status;
	  END_IF;
	  
	  
	  // LReal Flags
	  #instLKinCtrl_ValueFlagCtrl(activeCmdNo              := #statActiveCmdNo,
	                              activePathDataIdentifier := #instLKinCtrl_MC_ExecuteKinMotionCmd.activePathDataIdentifier,
	                              activePathDataName       := #instLKinCtrl_MC_ExecuteKinMotionCmd.activePathDataName,
	                              remainingDistanceActCmd  := #statRemainingDistanceActCmd,
	                              kinematicsStatusWord     := #tempKinematicsStatusWord,
	                              movePathStatus           := #statStatus,
	                              flagsBuffer              := #statFlagsBuffer,
	                              waitMain                 => #statWaitValueMain,
	                              valueFlags               := #valueFlags,
	                              waitFlags                := #statWaitValueFlags);
	  
	  // Check if flag control FB has thrown an error
	  IF #instLKinCtrl_ValueFlagCtrl.error THEN
	    #statStatus := #ERR_VALUE_FLAG_CONTROL;
	    #statSubfunctionStatus := #instLKinCtrl_ValueFlagCtrl.status;
	  END_IF;
	  
	  // Save written active cmd number for "ExecuteKinMotionCmd" input
	  #statWrittenActiveCmdNo := #statActiveCmdNo;
	END_REGION FLAG_HANDLING
	
	//Reset preprocessing stop
	IF #statMCExecuteWasDone = TRUE //Execution of commands is done
	  AND #statWaitMain = FALSE
	  AND #statWaitValueMain = FALSE
	  AND #statPathDataElementPreBuffered.cmdID = #instLKinCtrl_MC_ExecuteKinMotionCmd.activeCmdNo
	THEN
	  #instLKinCtrl_PreBuffer.preprocessingStop := FALSE;
	END_IF;
	
	REGION OUTPUTS
	  // Write outputs
	  IF (#statStatus = #STATUS_EXECUTION_FINISHED) AND (#statDone = FALSE) THEN // Execution finished without errors
	    #statDone := TRUE;
	    #statBusy := FALSE;
	    #statCommandAborted := FALSE;
	    #statError := FALSE;
	    #statStateExecution := #EX_NO_PROCESSING; // Switch state machine to "no processing"
	    
	  ELSIF (#statStatus.%X15 = TRUE) AND (#statError = FALSE) THEN // Error occurred (#statStatus is 16#8000 to 16#FFFF)
	    #statDone := FALSE;
	    #statBusy := FALSE;
	    #statCommandAborted := FALSE;
	    #statError := TRUE;
	    // Write diagnostics
	    #diagnostics.statusSubFunction := #statSubfunctionStatus;
	    #statStateExecution := #EX_ERROR_STATE; // Switch state machine to "no processing"
	    
	  ELSIF (#statStatus = #STATUS_COMMAND_ABORTED) AND (#statCommandAborted = FALSE) THEN // Commanded functionality has been aborted by another command
	    #statDone := FALSE;
	    #statBusy := FALSE;
	    #statCommandAborted := TRUE;
	    #statError := FALSE;
	    // Write diagnostics
	    #diagnostics.statusSubFunction := #statSubfunctionStatus;
	    #statStateExecution := #EX_NO_PROCESSING; // Switch state machine to "no processing"
	    
	  ELSIF (#tempExecute = FALSE) AND (#tempStop = FALSE) AND ((#statDone = TRUE) OR (#statError = TRUE) OR (#statCommandAborted = TRUE)) THEN // Reset outputs
	    #statDone := FALSE;
	    #statBusy := FALSE;
	    #statCommandAborted := FALSE;
	    #statError := FALSE;
	    #statReadyForNextPath := TRUE; // Added FR 2019/04/11
	    #statStatus := #STATUS_NO_CALL;
	    #statActivePathData := '';
	    #statActiveCmdNo := 0;
	    #statRemainingDistanceActCmd := 0.0;
	  END_IF;
	  
	  // ------------------------------
	  // Write static values to outputs
	  // ------------------------------
	  #done := #statDone;
	  #busy := #statBusy;
	  #commandAborted := #statCommandAborted;
	  #error := #statError;
	  #status := #statStatus;
	  #readyForNextPath := #statReadyForNextPath;
	  #active := #instLKinCtrl_MC_ExecuteKinMotionCmd.active;
	  #activePathData := #statActivePathData;
	  #activeCmdNo := #statActiveCmdNo;
	  #remainingDistanceActCmd := #statRemainingDistanceActCmd;
	  
	  // ------------------------------
	  // Write diagnostics
	  // ------------------------------
	  IF #statError THEN
	    #diagnostics.errorID := #statStatus; // write status to errorID in case of error pending
	  END_IF;
	  
	  // Write status in every cycle
	  #diagnostics.stateMovePath := #statStateExecution;
	  #diagnostics.kinematicsStatusWord := #instLKinCtrl_MC_ExecuteKinMotionCmd.diagnostics.kinematicsStatusWord;
	END_REGION OUTPUTS
	
	// =================================================================================================================
	// End of Function Block: LKinCtrl_MC_MovePath
	// =================================================================================================================
END_FUNCTION_BLOCK

FUNCTION_BLOCK "LKinCtrl_SetFlagCtrl"
TITLE = LKinCtrl_SetFlagCtrl
{ S7_Optimized_Access := 'TRUE' }
AUTHOR : 'handling.team.automation@siemens.com'
FAMILY : LKinCtrl
VERSION : 5.0
//Handle setFlags in FB MovePath
   VAR_INPUT 
      enable { ExternalAccessible := 'False'; ExternalVisible := 'False'; ExternalWritable := 'False'} : Bool;   // TRUE: Enable functionality of FB
      activeCmdNo { ExternalAccessible := 'False'; ExternalVisible := 'False'; ExternalWritable := 'False'} : DInt;   // Number of actual PathData set number (interconnect LKinCtrl_MC_ExecuteKinMotionCmd)
      activePathDataIdentifier { ExternalAccessible := 'False'; ExternalVisible := 'False'; ExternalWritable := 'False'} : USInt;   // Identifier number of actual PathData (interconnect LKinCtrl_MC_ExecuteKinMotionCmd)
      activePathDataName { ExternalAccessible := 'False'; ExternalVisible := 'False'; ExternalWritable := 'False'} : String["LKINCTRL_LENGTH_OF_PATHDATA_NAME"];   // Name of actual PathData (interconnect LKinCtrl_MC_ExecuteKinMotionCmd)
      remainingDistanceActCmd { ExternalAccessible := 'False'; ExternalVisible := 'False'; ExternalWritable := 'False'} : LReal;   // RemainingDistance of active motionCommand (interconnect LKinCtrl_MC_ExecuteKinMotionCmd)
      kinematicsStatusWord { ExternalAccessible := 'False'; ExternalVisible := 'False'; ExternalWritable := 'False'} : DWord;   // Interconnect axesGroup.StatusWord
      movePathStatus { ExternalAccessible := 'False'; ExternalVisible := 'False'; ExternalWritable := 'False'} : Word;   // Interconnect value for MovePath output 'status'
      flagsBuffer { ExternalAccessible := 'False'; ExternalVisible := 'False'; ExternalWritable := 'False'} : Struct   // Buffer to store flag information for past and actual commands
         writeBufferElement { ExternalAccessible := 'False'; ExternalVisible := 'False'; ExternalWritable := 'False'} : Int := 1;   // pointer on entry to be written
         bufferElement { ExternalAccessible := 'False'; ExternalVisible := 'False'; ExternalWritable := 'False'} : Array[1.."LKINCTRL_NO_OF_SETFLAGS_BUFFER_ELEMENTS"] of Struct   // flag information for one specific command (see cmdId)
            pathDataName { ExternalAccessible := 'False'; ExternalVisible := 'False'; ExternalWritable := 'False'} : String["LKINCTRL_LENGTH_OF_PATHDATA_NAME"] := '';   // PathData name of specific command
            pathDataIdentifier { ExternalAccessible := 'False'; ExternalVisible := 'False'; ExternalWritable := 'False'} : DInt;   // PathData identifier counter of specific command
            cmdId { ExternalAccessible := 'False'; ExternalVisible := 'False'; ExternalWritable := 'False'} : DInt := 0;   // cmdId of command in PathData
            isIntermediateCmd { ExternalAccessible := 'False'; ExternalVisible := 'False'; ExternalWritable := 'False'} : Bool;   // TRUE: command is intermediate command
            setFlags { ExternalAccessible := 'False'; ExternalVisible := 'False'; ExternalWritable := 'False'} : Array[1.."LKINCTRL_NO_OF_CMD_SETFLAGS"] of "LKinCtrl_typeSetFlagElement_Bool";   // setFlags structure equal to PathData command entry
            valueFlags { ExternalAccessible := 'False'; ExternalVisible := 'False'; ExternalWritable := 'False'} : Array[1.."LKINCTRL_NO_OF_CMD_VALUEFLAGS"] of "LKinCtrl_typeSetFlagElement_LReal";   // setFlags structure equal to PathData command entry
         END_STRUCT;
      END_STRUCT;
   END_VAR

   VAR_OUTPUT 
      valid { ExternalWritable := 'False'} : Bool;   // TRUE: Valid set of output values available at the FB
      busy { ExternalWritable := 'False'} : Bool;   // TRUE: FB is not finished and new output values can be expected
      error { ExternalWritable := 'False'} : Bool;   // TRUE: An error occurred during the execution of the FB
      status { ExternalWritable := 'False'} : Word := #STATUS_NO_CALL;   // 16#0000 - 16#7FFF: Status of the FB, 16#8000 - 16#FFFF: Error identification
      waitMain { ExternalWritable := 'False'} : Bool;   // Static bit to wait for execution due to wait flags & valueFlags
   END_VAR

   VAR_IN_OUT 
      flags : Array[*] of Bool;   // Interconnect MovePath outputs for flag signals
      waitFlags : Struct   // Static struct to store wait flag information
         waitCtr : Int;   // counter for number of wait flags in one command
         waitFlag : Array[1.."LKINCTRL_NO_OF_CMD_SETFLAGS"] of Int;   // flag number as identifier for flag active as wait flag
      END_STRUCT;
   END_VAR

   VAR 
      statEnableOld { ExternalAccessible := 'False'; ExternalVisible := 'False'; ExternalWritable := 'False'} : Bool;   // Old value of 'enable' input for edge detection
      statValid { ExternalAccessible := 'False'; ExternalVisible := 'False'; ExternalWritable := 'False'} : Bool;   // Static value for output 'valid'
      statBusy { ExternalAccessible := 'False'; ExternalVisible := 'False'; ExternalWritable := 'False'} : Bool;   // Static value for output 'busy'
      statError { ExternalAccessible := 'False'; ExternalVisible := 'False'; ExternalWritable := 'False'} : Bool;   // Static value for output 'error'
      statErrorUserCleared { ExternalAccessible := 'False'; ExternalVisible := 'False'; ExternalWritable := 'False'} : Bool;   // Error occurred that can only be solved by user; rising edge at enable input necessary
      statErrorAutoCleared { ExternalAccessible := 'False'; ExternalVisible := 'False'; ExternalWritable := 'False'} : Bool;   // Error occurred that can be acknowledged by FB
      statStatus { ExternalAccessible := 'False'; ExternalVisible := 'False'; ExternalWritable := 'False'} : Word := #STATUS_NO_CALL;   // Static value for output 'status'
      statMovePathStatusOld { ExternalAccessible := 'False'; ExternalVisible := 'False'; ExternalWritable := 'False'} : Word;   // Static value for last status of MovePath
      statFBState { ExternalAccessible := 'False'; ExternalVisible := 'False'; ExternalWritable := 'False'} : DInt := #FB_STATE_NO_PROCESSING;   // State in the state machine of the FB
      statDisablingCompleted { ExternalAccessible := 'False'; ExternalVisible := 'False'; ExternalWritable := 'False'} : Bool;   // TRUE: Disabling has been completed
      statWaitMain { ExternalAccessible := 'False'; ExternalVisible := 'False'; ExternalWritable := 'False'} : Bool;   // Static value for output 'waitMain'
      statSkippedCmdCounter { ExternalAccessible := 'False'; ExternalVisible := 'False'; ExternalWritable := 'False'} : Int;   // Static counter for skipped activeCmdNo
      statActivePathDataIdentifierOld { ExternalAccessible := 'False'; ExternalVisible := 'False'; ExternalWritable := 'False'} : USInt;   // Static to store old activePathDataIdentifier from LKinCtrl_ExecuteKinMotionCmd
      statActiveCmdNoOld { ExternalAccessible := 'False'; ExternalVisible := 'False'; ExternalWritable := 'False'} : DInt;   // Static variable storing old 'activeCmdNo'
      statActivePathDataNameOld { ExternalAccessible := 'False'; ExternalVisible := 'False'; ExternalWritable := 'False'} : String["LKINCTRL_LENGTH_OF_PATHDATA_NAME"];   // Static to store last active PathData name
      statFlagSetAfterCmd { ExternalAccessible := 'False'; ExternalVisible := 'False'; ExternalWritable := 'False'} : Array[1.."LKINCTRL_NO_OF_CMD_SETFLAGS"] of Int;   // Static array storing flags to be set after command
      statWaitFlagSetAfterCmd { ExternalAccessible := 'False'; ExternalVisible := 'False'; ExternalWritable := 'False'} : Array[1.."LKINCTRL_NO_OF_CMD_SETFLAGS"] of Int;   // Static array storing wait flags to be set after command
      statFlagResetAfterOneCmd { ExternalAccessible := 'False'; ExternalVisible := 'False'; ExternalWritable := 'False'} : Array[1.."LKINCTRL_NO_OF_CMD_SETFLAGS"] of Int;   // Static array storing flags to be reset after one command
      statFlagResetFM3 { ExternalAccessible := 'False'; ExternalVisible := 'False'; ExternalWritable := 'False'} : Array[1.."LKINCTRL_NO_OF_CMD_SETFLAGS"] of Int;   // Static array storing flags to be reset after one cycle
      statFlagSetFM10 { ExternalAccessible := 'False'; ExternalVisible := 'False'; ExternalWritable := 'False'} : Array[1.."LKINCTRL_NO_OF_CMD_SETFLAGS"] of Int;   // Static array storing flags to be set at remaining distance
      statFlagResetFM10 { ExternalAccessible := 'False'; ExternalVisible := 'False'; ExternalWritable := 'False'} : Array[1.."LKINCTRL_NO_OF_CMD_SETFLAGS"] of Int;   // Static array storing flags to be reset at remaining distance
      statRemDistanceFM10 { ExternalAccessible := 'False'; ExternalVisible := 'False'; ExternalWritable := 'False'} : Array[1.."LKINCTRL_NO_OF_CMD_SETFLAGS"] of LReal;   // Static array storing remaining distance for flags
      statFlagSetFM13 { ExternalAccessible := 'False'; ExternalVisible := 'False'; ExternalWritable := 'False'} : Array[1.."LKINCTRL_NO_OF_CMD_SETFLAGS"] of Int;   // Static array storing flags to be set after command for one cycle
      statFlagResetFM13 { ExternalAccessible := 'False'; ExternalVisible := 'False'; ExternalWritable := 'False'} : Array[1.."LKINCTRL_NO_OF_CMD_SETFLAGS"] of Int;   // Static array storing flags to be set after command and reset after one cycle
      statWaitFlagActiveCmdId { ExternalAccessible := 'False'; ExternalVisible := 'False'; ExternalWritable := 'False'} : Array[1.."LKINCTRL_NO_OF_CMD_SETFLAGS"] of DInt;   // Static array storing active command number for watiFlag
      statWaitFlagActivePathData { ExternalAccessible := 'False'; ExternalVisible := 'False'; ExternalWritable := 'False'} : Array[1.."LKINCTRL_NO_OF_CMD_SETFLAGS"] of DInt;   // Static array storing active PathData number for watiFlag
      statFlagResetSkipped { ExternalAccessible := 'False'; ExternalVisible := 'False'; ExternalWritable := 'False'} : Array[1..#MAX_NUMBER_OF_SKIPPED_CMDS, 1.."LKINCTRL_NO_OF_CMD_SETFLAGS"] of Int;   // Static array storing flags to be reset after one cycle
      statWaitFlagOld { ExternalAccessible := 'False'; ExternalVisible := 'False'; ExternalWritable := 'False'} : Array[1.."LKINCTRL_NO_OF_CMD_SETFLAGS"] of Bool;   // Static array storing last flag values for reset detection
      statACKMode { ExternalAccessible := 'False'; ExternalVisible := 'False'; ExternalWritable := 'False'} : Array[1.."LKINCTRL_NO_OF_CMD_SETFLAGS"] of USInt;   // Static array storing acknowledge mode information
      statLowerBoundFlags { ExternalAccessible := 'False'; ExternalVisible := 'False'; ExternalWritable := 'False'} : DInt;
      statUpperBoundFlags { ExternalAccessible := 'False'; ExternalVisible := 'False'; ExternalWritable := 'False'} : DInt;
   END_VAR

   VAR_TEMP 
      tempEnable : Bool;   // Temporary value for input 'enable'
      tempFlagCmdCounter : Int;   // Temporary flag cmd counter for setFlag UDT
      tempFlagsBufferElementCtr : Int;   // Temporary flag buffer counter
      tempFlagCounter : Int;   // Temporary flag counter for flag array
      tempFlagWasSet : Bool;   // Temporary bool to signalize flag was set after end of PRG
      tempSkippedCounterInc : Bool;   // Temporary bool to signalize skipped counter was increased
   END_VAR

   VAR CONSTANT 
      FB_STATE_NO_PROCESSING : DInt := 0;   // FB state: No processing
      FB_STATE_CHECK_ACTIVE_CMD : DInt := 50;   // FB state: Check change of active command
      FB_STATE_SET_RESET_AFTER_COMMAND : DInt := 51;   // FB state: Handle flag actions after commands
      FB_STATE_EVALUATE_FLAGBUFFER : DInt := 52;   // FB state: Handle flagBuffer and flag actions before command
      FB_STATE_RESET_AFTER_ONE_CYCLE : DInt := 53;   // FB state: Handle flag reset after one cycle
      FB_STATE_CHECK_REMAINING_DISTANCE : DInt := 54;   // FB state: Check flag with remaining distance
      FB_STATE_WAIT_FLAG_HANDLING : DInt := 55;   // FB state: Check wait flags
      FB_STATE_DISABLING : DInt := 90;   // FB state: Disabling
      STATUS_NO_CALL : Word := 16#7000;   // No job being currently processed
      STATUS_FIRST_CALL : Word := 16#7001;   // First call after incoming new job (rising edge 'execute')
      STATUS_SUBSEQUENT_CALL : Word := 16#7002;   // Subsequent call during active processing without further details
      ERR_UNDEFINED_STATE : Word := 16#8600;   // Error due to an undefined state in state machine
      ERR_OVERFLOW_SKIPPED_CMDS : Word := 16#8601;   // Error due to overflow of skipped commands counter
      STATUS_EXECUTION_WAITING : Word := 16#7307;   // Status path execution waiting due to wait flag, wait time or single step mode
      MAX_NUMBER_OF_SKIPPED_CMDS : Int := 3;   // Maximum number of activeCmdNo to be skipped
   END_VAR


BEGIN
	//==========================================================================================
	// SIEMENS AG
	// (c)Copyright 2020 All Rights Reserved
	//------------------------------------------------------------------------------------------
	// Library: LKinCtrl
	// Tested with: S7-1517T-3 PN/DP
	// Engineering: TIA Portal V15
	// Restrictions: ---
	// Requirements: S7-1500T FW 2.5
	// Functionality: LKinCtrl_SetFlagCtrl
	// The FC evaluates the flag informaton given by the PathData structure and controls the flag
	// variables depending on the active command information given
	//
	// Support: tech.team.motioncontrol@siemens.com
	// Note: Parameter comments are only available in language 'English (United States)'
	//------------------------------------------------------------------------------------------
	// Change log table:
	// Version    Date          Expert in charge    Changes applied
	// 01.00.00   19.08.2019    JR                  First release version v1.0
	// 01.00.01   18.09.2019    JR                  Updates for LREAL flags
	// 01.00.02   19.09.2019    JR                  Implementation wait value flags - flagMode 5
	// 01.00.03   19.09.2019    JR                  Implementation value flags - flagMode 11 - 15
	// 01.00.04   27.11.2019    JR                  Additional condition for deactivating flags
	// 01.01.00   28.11.2019    JR                  Separate block for setFlags from LKinCtrl_FlagCtrl
	// 01.01.01   27.01.2020    FR                  Changed FM 10 from > to >=
	// 01.01.02   30.01.2020    FR                  Changed flag array constant
	// 02.00.00   12.03.2020    FR                  Reworked complete FB to fit enable template with state machine
	// 02.00.01   17.03.2020    FR                  Check remDistance <= 0.0 instead of =
	// 02.00.02   03.08.2020    FR                  Change interface actualCmdIsCircularCmd to KinematicsStatusWord (DWord)
	// 02.00.03   19.10.2020    FR                  Handle multiple commands per cycle; Changed case to use constants instead of numbers
	// 02.00.04   15.12.2020    FR                  Added option for SPTP commands to have calculated remainingDistance
	// 02.00.05   01.06.2021    FR                  Use variable instead of F_Trig, Fix for FM5 / FM15, Fix for statActiveCmdNoOld not being reset correctly
	// 02.00.06   29.10.2021    FR                  Added option to disable flag reset, added new FM25 & FM26
	// 02.00.07   04.01.2024    SF                  Added remaining distance check for MC_MovePickAndPlaceLinear integration
	//===========================================================================================
	
	#tempEnable := #enable; // Work with temporary value / create process image
	
	REGION ENABLING/DISABLING
	    IF (#tempEnable = TRUE) AND (#statStatus = #STATUS_NO_CALL) THEN // Enable FB
	        // First call; initialize FB
	        #statValid := TRUE;
	        #statBusy := TRUE;
	        #statError := FALSE;
	        #statErrorUserCleared := FALSE;
	        #statErrorAutoCleared := FALSE;
	        #statStatus := #STATUS_FIRST_CALL;
	        
	        #statLowerBoundFlags := LOWER_BOUND(ARR := #flags, DIM := 1);
	        #statUpperBoundFlags := UPPER_BOUND(ARR := #flags, DIM := 1);
	        
	        #statFBState := #FB_STATE_CHECK_ACTIVE_CMD; // State machine - start functionality
	        //------------------------------------------------------------------------------------------
	        // Initialize functionality: reset of variables, diagnostics, etc.
	        #statDisablingCompleted := FALSE;
	        
	        IF "LKINCTRL_DISABLE_FLAG_RESET" THEN
	            ;// no reset
	        ELSE
	            // Initialize all setFlags (flag array) when enabling
	            //------------------------------------------------------------------------------------------
	          FOR #tempFlagCounter := #statLowerBoundFlags TO #statUpperBoundFlags DO
	                #flags[#tempFlagCounter] := FALSE;
	            END_FOR;
	        END_IF;
	        
	        // Initialize flag handling variables
	        //------------------------------------------------------------------------------------------
	        // reset wait output
	        #statWaitMain := FALSE;
	        #statSkippedCmdCounter := 0;
	        #statActiveCmdNoOld := 0;
	        #statActivePathDataNameOld := '';
	        #statActivePathDataIdentifierOld := 0;
	        #statMovePathStatusOld := 16#0;
	        
	        FOR #tempFlagCmdCounter := 1 TO "LKINCTRL_NO_OF_CMD_SETFLAGS" DO
	            // reset auxiliary flag storage variables
	            #statFlagResetAfterOneCmd[#tempFlagCmdCounter] := -1;
	            #statFlagSetAfterCmd[#tempFlagCmdCounter] := -1;
	            #statWaitFlagSetAfterCmd[#tempFlagCmdCounter] := -1;
	            #statFlagResetFM3[#tempFlagCmdCounter] := -1;
	            #statFlagResetFM10[#tempFlagCmdCounter] := -1;
	            #statFlagResetFM13[#tempFlagCmdCounter] := -1;
	            #statFlagSetFM13[#tempFlagCmdCounter] := -1;
	            #statFlagSetFM10[#tempFlagCmdCounter] := -1;
	            #statRemDistanceFM10[#tempFlagCmdCounter] := 0.0;
	            #statWaitFlagActiveCmdId[#tempFlagCmdCounter] := 0;
	            #statWaitFlagActivePathData[#tempFlagCmdCounter] := 0;
	            
	            #statACKMode[#tempFlagCmdCounter] := 0;
	            
	            // Initialize functionality: call subsidiary FBs with FALSE
	            #statWaitFlagOld[#tempFlagCmdCounter] := FALSE;
	            
	            // Reset storage for skipped commands
	            FOR #tempFlagCounter := 1 TO #MAX_NUMBER_OF_SKIPPED_CMDS DO
	                #statFlagResetSkipped[#tempFlagCounter, #tempFlagCmdCounter] := -1;
	            END_FOR;
	        END_FOR;
	        
	        
	        //------------------------------------------------------------------------------------------
	        
	    ELSIF (#tempEnable = FALSE) AND (#statEnableOld = TRUE) THEN // Disable FB 
	        #statFBState := #FB_STATE_DISABLING;
	        
	    ELSIF (#statStatus = #STATUS_FIRST_CALL) THEN // Set status identifier of subsequent call
	        #statStatus := #STATUS_SUBSEQUENT_CALL;
	    END_IF;
	    
	    // Edge detection 'enable' input
	    #statEnableOld := #tempEnable;
	END_REGION ENABLING/DISABLING
	
	IF (#statStatus = #STATUS_NO_CALL) THEN // Nothing to do -> End here to reduce "system load"
	    RETURN;
	END_IF;
	
	REGION STATE_MACHINE
	    // Use if sate machine for more states in one cycle
	    
	    // No processing active (Note: this state must always be present and left empty)
	    IF #statFBState = #FB_STATE_NO_PROCESSING THEN
	        ;
	    END_IF;
	    
	    // Reset after one cycle 
	    REGION STATE_RESET_AFTER_ONE_CYCLE
	        IF #statFBState = #FB_STATE_RESET_AFTER_ONE_CYCLE THEN
	            // for loop checking all available flags
	            FOR #tempFlagCmdCounter := 1 TO "LKINCTRL_NO_OF_CMD_SETFLAGS" DO
	                // reset flags active for one cycle only (flagMode: 3)
	                IF #statFlagResetFM3[#tempFlagCmdCounter] <> -1 THEN
	                    // reset flags when active command is ended / next command starts
	                    #flags[#statFlagResetFM3[#tempFlagCmdCounter]] := FALSE;
	                    // reset stored flag to be reset (to not reset it after each single future command)
	                    #statFlagResetFM3[#tempFlagCmdCounter] := -1;
	                END_IF;
	                
	                // reset flags active for one cycle only (flagMode: 13)
	                IF #statFlagResetFM13[#tempFlagCmdCounter] <> -1 THEN
	                    // reset flags when active command is ended / next command starts
	                    #flags[#statFlagResetFM13[#tempFlagCmdCounter]] := FALSE;
	                    // reset stored flag to be reset (to not reset it after each single future command)
	                    #statFlagResetFM13[#tempFlagCmdCounter] := -1;
	                END_IF;
	                
	                // Check if commands were skipped and reset flags
	                FOR #tempFlagCounter := 1 TO #statSkippedCmdCounter DO // If no cmd was skipped the upper limit should be 0 --> No execution of the loop
	                    // If activeCmdNo was skipped reset flags active for one cycle only (flagMode: 2/3/13)
	                    IF #statFlagResetSkipped[#tempFlagCounter, #tempFlagCmdCounter] <> -1 THEN
	                        // reset flags when active command is ended / next command starts
	                        #flags[#statFlagResetSkipped[#tempFlagCounter, #tempFlagCmdCounter]] := FALSE;
	                        // reset stored flag to be reset (to not reset it after each single future command)
	                        #statFlagResetSkipped[#tempFlagCounter, #tempFlagCmdCounter] := -1;
	                    END_IF;
	                END_FOR;
	            END_FOR;
	            
	            // go to next state
	            #statFBState := #FB_STATE_CHECK_ACTIVE_CMD;
	        END_IF;
	    END_REGION STATE_RESET_AFTER_ONE_CYCLE
	    
	    
	    // Cyclic state
	    // This state shall be the idle state where conditions are checked 
	    // --> Change in active command number
	    // --> End of cmd
	    // --> End of prg
	    // --> ...
	    REGION STATE_CHECK_ACTIVE_CMD
	        IF #statFBState = #FB_STATE_CHECK_ACTIVE_CMD THEN // Processing active
	            // Check if activeCmdNo has changed or MovePath is waiting and remainingDistance = 0
	            // --> Go to state: #FB_STATE_SET_RESET_AFTER_COMMAND
	            // Else
	            // --> Go to state: #FB_STATE_CHECK_REMAINING_DISTANCE
	            //
	            // Check if active cmd no has changed // changed JR 2019/04/11 < to <>
	            IF (#statActiveCmdNoOld <> #activeCmdNo OR #statActivePathDataIdentifierOld <> #activePathDataIdentifier)
	                OR (#movePathStatus = #STATUS_EXECUTION_WAITING AND #remainingDistanceActCmd <= 0.0) // check for command to be finished
	                OR (#movePathStatus <> 16#730A AND #statMovePathStatusOld = 16#730A) // end of configuration command
	            THEN
	                #statFBState := #FB_STATE_SET_RESET_AFTER_COMMAND;
	            ELSE
	                #statFBState := #FB_STATE_CHECK_REMAINING_DISTANCE;
	            END_IF;
	        END_IF;
	    END_REGION STATE_CHECK_ACTIVE_CMD
	    
	    
	    // Set / Reset flags after command has finished (FM2 / FM11 / FM13 / FM15)
	    REGION STATE_SET_RESET_AFTER_COMMAND
	        IF #statFBState = #FB_STATE_SET_RESET_AFTER_COMMAND THEN
	            // for loop checking all available flags
	            FOR #tempFlagCmdCounter := 1 TO "LKINCTRL_NO_OF_CMD_SETFLAGS" DO
	                // reset flags active for one command only (flagMode: 2 (LKINCTRL_FM_SET_BEFORE_AND_RESET_AFTER))
	                IF #statFlagResetAfterOneCmd[#tempFlagCmdCounter] <> -1 THEN
	                    // reset flags when active command is ended / next command starts
	                    #flags[#statFlagResetAfterOneCmd[#tempFlagCmdCounter]] := FALSE;
	                    // reset stored flag to be reset (to not reset it after each single future command)
	                    #statFlagResetAfterOneCmd[#tempFlagCmdCounter] := -1;
	                END_IF;
	                
	                // set flags to be activated at end of command
	                // flagMode: 11 (LKINCTRL_FM_SET_AFTER_AND_NO_RESET)
	                IF #statFlagSetAfterCmd[#tempFlagCmdCounter] <> -1 THEN
	                    // set flags when active command is ended / next command starts
	                    #flags[#statFlagSetAfterCmd[#tempFlagCmdCounter]] := TRUE;
	                    // reset stored flag to be set (to not set it after each single future command)
	                    #statFlagSetAfterCmd[#tempFlagCmdCounter] := -1;
	                END_IF;
	                
	                // flagMode: 15 (LKINCTRL_FM_SET_AFTER_AND_NO_RESET_AND_WAIT_FOR_ACKNOWLEDGE)
	                IF #statWaitFlagSetAfterCmd[#tempFlagCmdCounter] <> -1 THEN
	                    // set flags when active command is ended / next command starts
	                    #flags[#statWaitFlagSetAfterCmd[#tempFlagCmdCounter]] := TRUE;
	                    #statWaitFlagOld[#tempFlagCmdCounter] := TRUE;
	                    // reset stored flag to be set (to not set it after each single future command)
	                    #statWaitFlagSetAfterCmd[#tempFlagCmdCounter] := -1;
	                END_IF;
	                
	                // set flags to be activated at end of command
	                // flagMode: 13 (LKINCTRL_FM_SET_AFTER_AND_RESET_AFTER_ONE_CYCLE)
	                IF #statFlagSetFM13[#tempFlagCmdCounter] <> -1 THEN
	                    // set flags when active command is ended / next command starts
	                    #flags[#statFlagSetFM13[#tempFlagCmdCounter]] := TRUE;
	                    
	                    // Save flag numbers to be reset after one cycle
	                    #statFlagResetFM13[#tempFlagCmdCounter] := #statFlagSetFM13[#tempFlagCmdCounter];
	                    
	                    // reset stored flag to be set (to not set it after each single future command)
	                    #statFlagSetFM13[#tempFlagCmdCounter] := -1;
	                END_IF;
	                
	                // Check if FM10 was not executed and set if next command is reached
	                IF (#statFlagSetFM10[#tempFlagCmdCounter] <> -1) THEN
	                    // Set flag if remaining distance is reached
	                    #flags[#statFlagSetFM10[#tempFlagCmdCounter]] := TRUE;
	                    // reset stored flag to be reset (to not reset it after each single future command)
	                    #statFlagSetFM10[#tempFlagCmdCounter] := -1;
	                    #statRemDistanceFM10[#tempFlagCmdCounter] := 0.0;
	                END_IF;
	                
	            END_FOR;
	            
	            // go to next state ; skip new flag if waiting
	            IF #movePathStatus = #STATUS_EXECUTION_WAITING
	                AND NOT (#statActiveCmdNoOld <> #activeCmdNo OR #statActivePathDataIdentifierOld <> #activePathDataIdentifier)
	            THEN
	                #statFBState := #FB_STATE_CHECK_REMAINING_DISTANCE;
	            ELSE
	                #statFBState := #FB_STATE_EVALUATE_FLAGBUFFER;
	            END_IF;
	        END_IF;
	    END_REGION STATE_SET_RESET_AFTER_COMMAND
	    
	    // Set flags before command and save variables to set after command (STATE_SET_RESET_AFTER)
	    // This state shall be used to copy flag buffer into variables 
	    // This state is reached after the state to set/reset flags after a command 
	    // --> Set flags before command instantly 
	    // --> Set flags after command in next call because of the state machine order
	    REGION STATE_EVALUATE_FLAGBUFFER
	        IF #statFBState = #FB_STATE_EVALUATE_FLAGBUFFER THEN
	            // Reset counter
	            #statSkippedCmdCounter := 0;
	            
	            // Reset activeCmdNoOld when PathData changes
	            IF #activeCmdNo = 1 THEN
	                #statActiveCmdNoOld := 0;
	            END_IF;
	            
	            // only run flag controls when a set is active
	            IF #activeCmdNo > 0 THEN
	                // selection of active flags and evaluation of flagMode
	                FOR #tempFlagsBufferElementCtr := 1 TO "LKINCTRL_NO_OF_SETFLAGS_BUFFER_ELEMENTS" DO
	                    IF #flagsBuffer.bufferElement[#tempFlagsBufferElementCtr].pathDataIdentifier = #activePathDataIdentifier // choose correct setFlags stored according to corresponding PathData
	                        AND #flagsBuffer.bufferElement[#tempFlagsBufferElementCtr].cmdId <= #activeCmdNo // choose only flags to be controlled when corresponding command is active
	                        AND #flagsBuffer.bufferElement[#tempFlagsBufferElementCtr].cmdId > #statActiveCmdNoOld // Also check flags on previous commands
	                    THEN
	                        // Reset temp to allow skippedCmdCounter to be increased
	                        #tempSkippedCounterInc := FALSE;
	                        
	                        // set flags according to PathData configuration stored in #statStoreSetFlagsBuffer
	                        FOR #tempFlagCmdCounter := 1 TO "LKINCTRL_NO_OF_CMD_SETFLAGS" DO
	                            
	                            // check for flag not to be deactivated
	                            IF #flagsBuffer.bufferElement[#tempFlagsBufferElementCtr].setFlags[#tempFlagCmdCounter].flag > -1 THEN
	                                
	                                CASE #flagsBuffer.bufferElement[#tempFlagsBufferElementCtr].setFlags[#tempFlagCmdCounter].flagMode OF
	                                        //------------------------------------------------------------------------------------------
	                                    "LKINCTRL_FM_SET_BEFORE_AND_NO_RESET": // FM 1
	                                        // (activate flag at beginning of command)
	                                        // set selected flag to TRUE at beginning of command
	                                        #flags[#flagsBuffer.bufferElement[#tempFlagsBufferElementCtr].setFlags[#tempFlagCmdCounter].flag] := TRUE;
	                                        //------------------------------------------------------------------------------------------
	                                        
	                                        //------------------------------------------------------------------------------------------
	                                    "LKINCTRL_FM_SET_BEFORE_AND_RESET_AFTER": // FM 2
	                                        // (activate flag at beginning of command)
	                                        // set selected flag to TRUE at beginning of command
	                                        #flags[#flagsBuffer.bufferElement[#tempFlagsBufferElementCtr].setFlags[#tempFlagCmdCounter].flag] := TRUE;
	                                        
	                                        IF #flagsBuffer.bufferElement[#tempFlagsBufferElementCtr].cmdId = #activeCmdNo THEN
	                                            // store flags to be set for one command only to reset at the end of command
	                                            #statFlagResetAfterOneCmd[#tempFlagCmdCounter] := #flagsBuffer.bufferElement[#tempFlagsBufferElementCtr].setFlags[#tempFlagCmdCounter].flag;
	                                        ELSE
	                                            // Check if skippedCmdCounter must be increased
	                                            IF NOT #tempSkippedCounterInc THEN
	                                                #statSkippedCmdCounter += 1;
	                                                #tempSkippedCounterInc := TRUE; // Store bit to avoid counting several times per command
	                                                IF #statSkippedCmdCounter > #MAX_NUMBER_OF_SKIPPED_CMDS THEN
	                                                    // Throw error
	                                                    #statStatus := #ERR_OVERFLOW_SKIPPED_CMDS;
	                                                    #statErrorUserCleared := TRUE;
	                                                    EXIT;
	                                                END_IF;
	                                            END_IF;
	                                            // ActiveCmdNo was skipped --> Store flag number to be reset after one cycle
	                                            #statFlagResetSkipped[#statSkippedCmdCounter, #tempFlagCmdCounter] := #flagsBuffer.bufferElement[#tempFlagsBufferElementCtr].setFlags[#tempFlagCmdCounter].flag;
	                                        END_IF;
	                                        //------------------------------------------------------------------------------------------
	                                        
	                                        //------------------------------------------------------------------------------------------
	                                    "LKINCTRL_FM_SET_BEFORE_AND_RESET_AFTER_ONE_CYCLE": // FM 3
	                                        // (activate flag at beginning of command for one cycle only)
	                                        // set selected flag to TRUE at beginning of command
	                                        #flags[#flagsBuffer.bufferElement[#tempFlagsBufferElementCtr].setFlags[#tempFlagCmdCounter].flag] := TRUE;
	                                        
